TYPE DUT_TEST :
STRUCT
	TEST01: UINT;
	TEST02: REAL;
END_STRUCT
END_TYPE

(* stored: Version 1.1.0.1, ProductVersion 3.1.4024.4
   DUT DUT_TEST: Id {3996e2ec-56a8-40c6-bda2-a07d646cc0f6} *)
